(* PLC project box, Dassault Systèmes ControlBuild 2024x *)
(* stored: creationDateTime 2023-10-03T11:13:33-01:00 *)

(* This module simulates a generic product "box". *)
FUNCTION_BLOCK equipment_library.box
  VAR
    status_act_prod : DINT := 0;
    m11 : REAL := 1.0;
    m12 : REAL := 0.0;
    m13 : REAL := 0.0;
    m14 : REAL := 0.0;
    m21 : REAL := 0.0;
    m22 : REAL := 1.0;
    m23 : REAL := 0.0;
    m24 : REAL := 0.0;
    m31 : REAL := 0.0;
    m32 : REAL := 0.0;
    m33 : REAL := 1.0;
    m34 : REAL := 0.0;
    m41 : REAL := 0.0;
    m42 : REAL := 0.0;
    m43 : REAL := 0.0;
    m44 : REAL := 1.0;
    movementConv : REAL := 0.0;
    contact : BOOL := false;
    centreRotX : REAL := 0.0;
    centreRotZ : REAL := 0.0;
    centreRotY : REAL := 0.0;
    moveDirection : INT := 0;
    idConv : DINT := 0;
    moveAuthorization : BOOL := false;
    number : INT := 0;
    idProdBelow : DINT := 0;
    oldOtherPx : REAL := 0.0;
    oldOtherPy : REAL := 0.0;
    oldOtherPz : REAL := 0.0;
    oldOtherRx : REAL := 0.0;
    oldOtherRy : REAL := 0.0;
    oldOtherRz : REAL := 0.0;
    gravitySpeed : REAL := 0.0;
    oldIdConv : DINT := 0;
  END_VAR


ACTION Prelude:
/* ----------------------------------------------------------------	*/
/* Initialisation of local variables of the instance of the product	*/
/* ----------------------------------------------------------------	*/

movementConv = 0.0;
contact = 0;
moveAuthorization = 1;
idConv=-1;
END_ACTION

ACTION Postlude:
/* ----------------------------------------------------------------	*/
/* If there is no contact, the box falls down thanks to gravity	*/	
/* ----------------------------------------------------------------	*/
if (contact == 0) 
	moveZBy(myself, gravitySpeed*-1.0);


/* ----------------------------------------------------------------	*/
/* Shift on conveyors if authorization					*/
/* ----------------------------------------------------------------	*/
if (moveAuthorization == 1 && (idConv>=0)) 
	moveRelativeAnotherBy(myself, idConv, movementConv, 0.0, 0.0);


/* ----------------------------------------------------------------	*/
/* Reset memories								*/
/* ----------------------------------------------------------------	*/
if (contact == 0) {
	moveDirection = 0;
	idProdBelow = -1;
}
END_ACTION

ACTION equipment_library.product_creator:
/* ----------------------------------------------------------------	*/
/* Information to the creation module that a product is in its area	*/
/* ----------------------------------------------------------------	*/
 
otherVar(productPresence) = 1;
END_ACTION

ACTION equipment_library.conveyor:
/* ----------------------------------------------------------------	*/
/* Interaction between the product and conveyors			*/
/* Convention : a conveyor is always oriented so that its X-axis is	*/
/*	  	  in the same direction as the flow			*/
/* ----------------------------------------------------------------	*/

/* ----------------------------------------------------------------	*/
/* We retrieve the conveyor's data if the center of the product is	*/
/* included in the volume of the conveyor.				*/
/* ----------------------------------------------------------------	*/
if ((idConv == -1) || isMyCenterIncludedInXYOfOther(myself, other)) {
	/* Traverse speed on the conveyor	*/
	movementConv = otherVar(incShiftProduct) ;

	/* Keep trace of traverse direction of the conveyor		*/
	if (movementConv  > 0.0) moveDirection = DIR_FLOW;
	if (movementConv  < 0.0) moveDirection = DIR_INVERSE_FLOW;

	/* Get the identifier of the conveyor in order to be		*/
	/* able to shift the product in its coordinate system		*/
	idConv = other;
	oldIdConv = idConv;

	/* If the conveyor is a traverser, a lift, ...  		*/
	/* the product msut follow it	 				*/
	if (otherVar(incrementPositionX) != 0.0) moveXBy(myself, otherVar(incrementPositionX));
	if (otherVar(incrementPositionY) != 0.0) moveYBy(myself, otherVar(incrementPositionY));
	if (otherVar(incrementPositionZ) != 0.0) alignTwoObjectsRelativeThirdZ(myself, other, other);

	/* Management of the rotation of the product on a 		*/
	/* swivelling table, rotary plate ring, ...			*/
	/* Keep trace of the rotation center in order to be 		*/
	/* able to give them to products that could be stacked		*/
	/* above this instance						*/
	centreRotX = otherVar(centerRotX);
	centreRotY = otherVar(centerRotY);
	centreRotZ = otherVar(centerRotZ);

	if ((otherVar(incRotX) != 0.0) || (otherVar(incRotY)!= 0) || (otherVar(incRotZ)!= 0.0))
		rotateBy(myself, otherVar(incRotX), otherVar(incRotY), otherVar(incRotZ), centreRotX, centreRotY, centreRotZ);  

}

/* ----------------------------------------------------------------	*/
/* The product lays on a solid						*/
/* ----------------------------------------------------------------	*/
contact = 1;
END_ACTION

ACTION equipment_library.stop:
/* ----------------------------------------------------------------	*/
/* Stop on a mechanical stop	  					*/
/* Management of the interaction with a mechanical stop with or 	*/
/* without blocking of the product on the mechanical stop according	*/
/* to the shift direction.							*/
/* ----------------------------------------------------------------	*/


/* The movement of the product can be forbidden according to the 	*/
/* position of the mechanical stop, the position of the product 	*/
/* and the shift direction. 						*/
if ( oldIdConv >= 0 && ((moveDirection == DIR_FLOW && (getCenterXInAnother(myself, oldIdConv ) < getCenterXInAnother(other, oldIdConv ))) 
	|| (moveDirection == DIR_INVERSE_FLOW && (getCenterXInAnother(myself, oldIdConv ) > getCenterXInAnother(other, oldIdConv )))) ) {

	moveAuthorization=0;
 }
END_ACTION

ACTION equipment_library.presence_sensor:
/* ----------------------------------------------------------------	*/
/* Information to the sensor that a product is in its detection area	*/
/* ----------------------------------------------------------------	*/

otherVar(detection) = 1;
END_ACTION

ACTION equipment_library.product_killer:
/* ----------------------------------------------------------------	*/
/* Destruction of the current instance of the product if the killer	*/
/* is active.									*/
/* ----------------------------------------------------------------	*/

if (otherVar(isActive)) prodKill(myself);
END_ACTION

ACTION equipment_library.suction_head:
/* ----------------------------------------------------------------	*/
/* Information to the actor that a product is present			*/
/* ----------------------------------------------------------------	*/
otherVar(productPresence) = 1;

/* ----------------------------------------------------------------	*/
/* Keep contact with the actor only if the head is sucking		*/
/* ----------------------------------------------------------------	*/
if (otherVar(suckProduct)) {
	moveRelativeAnotherBy(myself, other, otherVar(incrementPositionX), otherVar(incrementPositionY), otherVar(incrementPositionZ));
	contact = 1;
}
END_ACTION

ACTION equipment_library.box:
/* ----------------------------------------------------------------	*/
/* Interaction between two products	 				*/
/* ----------------------------------------------------------------	*/


/* Verify that the product whose position has to be updated is 	*/
/* located on one side of the current instance and not above or 	*/
/* below it.									*/
if ((getCenterZ(myself) > getCenterZ(other) - (getSizeZ(other)/2.0)) && (getCenterZ(myself) < getCenterZ(other)+(getSizeZ(other)/2.0))) {
	/* Update the position of the product that is behind the 	*/
	/* other according to the shift direction				*/
	if ( (moveDirection == DIR_FLOW && (getCenterXInAnother(myself, idConv) < getCenterXInAnother(other, idConv))) 
		|| (moveDirection == DIR_INVERSE_FLOW && (getCenterXInAnother(myself, idConv) > getCenterXInAnother(other, idConv))) ) {

		/* Align the 2 products one behind the other if its speed is lower 		*/
		if (fabs(movementConv ) > fabs(otherVar(movementConv )))
			alignTwoObjectsRelativeThirdX(myself, other, idConv);

		/* Forbid the shift						*/
		moveAuthorization=0;
	 }
}

/* Interaction with the product below					*/
if ((getCenterZ(myself)  > getCenterZ(other)+ (getSizeZ(other) / 2)) 
	&&  ((getCenterX(myself) > getCenterX(other) - (getSizeX(other)/4.0)) && (getCenterX(myself) < getCenterX(other)+(getSizeX(other)/4.0)))
	&&  ((getCenterY(myself) > getCenterY(other) - (getSizeY(other)/4.0)) && (getCenterY(myself) < getCenterY(other)+(getSizeY(other)/4.0))))  {
	/* Same movement than the product below				*/
	if (idProdBelow == other) {
		moveBy(myself, getPositionX(other)-oldOtherPx, getPositionY(other)-oldOtherPy, getPositionZ(other)-oldOtherPz);
		rotateBy(myself, getAngleX(other)-oldOtherRx, getAngleY(other)-oldOtherRy, getAngleZ(other)-oldOtherRz,
				otherVar(centreRotX), otherVar(centreRotY), otherVar(centreRotZ));
	}
	oldOtherPx=getPositionX(other); oldOtherPy=getPositionY(other); oldOtherPz=getPositionZ(other);
	oldOtherRx=getAngleX(other); oldOtherRy=getAngleY(other); oldOtherRz=getAngleZ(other);
	centreRotX=otherVar(centreRotX); centreRotY=otherVar(centreRotY); centreRotZ=otherVar(centreRotZ);

	idProdBelow = other;

	/* The product lays on a solid					*/
	contact = 1;

	/* The next line of code can be added in order to align 	*/
	/* correctly  the products one on the others ...		*/
	/* We should align both products in Z-axis according to the 	*/
	/* absolute coordinate system and not according to the 	*/
	/* relative system coordinate in order to have a generic 	*/
	/* behaviour.								*/
	/* => adapt this according to the application when needed	*/

	/* alignTwoObjectsRelativeThirdZ(myself, other, other); 	*/
	
}
END_ACTION

ACTION equipment_library.tipper:
/* ----------------------------------------------------------------	*/
/* The product turns over 							*/
/* ----------------------------------------------------------------	*/
if (otherVar(incrementRotation != 0.0)) {
	rotateYBy(myself, otherVar(incrementRotation),otherVar(initPosX),
		 otherVar(initPosY), otherVar(initPosZ));
	moveAuthorization = 0;
} 
else {
/* automatic repositionning of the product on fixed positions  */
	CB_Float fixedPositions[5]={0.0, 90.0, 180.0, 270.0, 360.0};
	CB_Float deltaRecalage = 10.0;
	CB_Int i;
	CB_Float currentAngle;
	currentAngle=getAngleY(myself);  
	for (i=0; i<5; i++) {
		if ((currentAngle- deltaRecalage < fixedPositions[i]) && (currentAngle+ deltaRecalage > fixedPositions[i])) {
			if (currentAngle!= fixedPositions[i]) {
				rotateYTo(myself, fixedPositions[i],otherVar(initPosX),otherVar(initPosY), otherVar(initPosZ));
			}
			break;
		 }
	}
}



/* ----------------------------------------------------------------	*/
/* The product lays on a solid						*/
/* ----------------------------------------------------------------	*/
contact = 1;
END_ACTION

ACTION C_header:
#define DIR_FLOW		1
#define DIR_INVERSE_FLOW	-1
END_ACTION
END_FUNCTION_BLOCK
